(* CODESYS project SLL_Common_exported_from_plc.library
   Title: SLL Common
   CompiledLibraryCompatibilityVersion: CODESYS V3.5 SP16 Patch 5
   DefaultNamespace: SLL_Common
   Version: 0.0.0.1
   Placeholder: SLL_Common
   Company: SLL

Project tree, tasks and I/O mapping:
  libraries: Util, 3.5.19.0 (System); Standard, 3.5.18.0 (System); SysTime, 3.5.17.0 (System); BASIC, 3.3.3.0 (OSCAT)
  Common Control/
    Convert/
    PID/
    Selectors/
    SCALING/
      Stuctures/
      Function Blocks/
      Functions/
  Common Control/
    PID/
      function block Control_PI_Basic [ST]
      data type PID_Settings_Basic
  Convert/
    Functions/
      function TIME_Dword_To_Secs [ST]
      function TIME_Dword_To_Mins [ST]
  SCALING/
    Stuctures/
      data type DUT_SENSOR_SCALE_DWORD_IN_REAL_OUT
      data type DUT_SENSOR_SCALE_REAL_IN_REAL_OUT
      data type DUT_SENSOR_SCALE_WORD_IN_REAL_OUT
      data type DUT_SENSOR_SCALE_DINT_TO_REAL
      data type Union_SensorStatusBits
      data type DUT_SensorStatusBits
    Function Blocks/
      function block Sensor_Scale_Real_To_Real_Struct [FBD]
      function block Sensor_Scale_Dint_To_Real [FBD]
    Functions/
  HMI/
    Functions/
      function HMI_Time_Remain_HHMMSS [ST]
      function HMI_Bool_To_Enable [ST]
      function HMI_Concat_Units [ST]
      function HMI_Sensor_Byte_String [ST]
  SIM/
    function block SIM_Bool [FBD]
    function block SIM_Uint [FBD]
    function block SIM_Byte [FBD]
    function block SIM_Real [FBD]
    function block SIM_Word [FBD]
  STATS/
    function block Cycle_Freq [FBD]
    function block Timestamp_TO [FBD]
    function block Operated_Time_Hours [FBD]
    function block Operated_Time_Min [FBD]
    function block Operated_Time_Sec [FBD]
    function block Cycle_Freq_REAL [FBD]
  SEL/
    function block SEL_Bumpless_Word [FBD]
    function block SEL_Bumpless_Real [FBD]
    function block SEL_Bumpless_Bool [FBD]
    function block SEL_Bumpless_Byte [FBD]
  TIMERS/
    function block DUTY_CYCLE [FBD]
  INPUT/
    function block SWITCH_DEBOUNCE [FBD]
*)

// Common Control/PID/PID_Settings_Basic
TYPE PID_Settings_Basic :
STRUCT
	SUP : REAL;
	OFS : REAL;
	KP : REAL;
	TN : REAL;
	TV : REAL;
	LL : REAL;
	LH : REAL;
	NAME:STRING(20);
END_STRUCT
END_TYPE

// SCALING/Stuctures/DUT_SENSOR_SCALE_DWORD_IN_REAL_OUT
TYPE DUT_SENSOR_SCALE_DWORD_IN_REAL_OUT :
STRUCT
	RAW_UNDER_RANGE:DWORD;	
	RAW_MIN:DWORD;
	RAW_MAX:DWORD;
	RAW_OVER_RANGE:DWORD;
	SCL_MIN:REAL;
	SCL_MAX:REAL;
	BYPASS:BOOL:=0;
	BYPASS_SCL:DWORD:=0;	
END_STRUCT
END_TYPE

// SCALING/Stuctures/DUT_SENSOR_SCALE_REAL_IN_REAL_OUT
TYPE DUT_SENSOR_SCALE_REAL_IN_REAL_OUT :
STRUCT
	RAW_UNDER_RANGE:REAL;	
	RAW_MIN:REAL;
	RAW_MAX:REAL;
	RAW_OVER_RANGE:REAL;
	SCL_MIN:REAL;
	SCL_MAX:REAL;
	BYPASS:BOOL:=0;
	BYPASS_SCL:REAL:=0;		
END_STRUCT
END_TYPE

// SCALING/Stuctures/DUT_SENSOR_SCALE_WORD_IN_REAL_OUT
TYPE DUT_SENSOR_SCALE_WORD_IN_REAL_OUT :
STRUCT
	RAW_UNDER_RANGE:WORD;	
	RAW_MIN:WORD;
	RAW_MAX:WORD;
	RAW_OVER_RANGE:WORD;
	SCL_MIN:REAL;
	SCL_MAX:REAL;
	BYPASS:BOOL:=0;
	BYPASS_SCL:WORD:=0;
	NAME: STRING(20);
	UNITS: STRING(10);
END_STRUCT
END_TYPE

// SCALING/Stuctures/DUT_SENSOR_SCALE_DINT_TO_REAL
TYPE DUT_SENSOR_SCALE_DINT_TO_REAL :
STRUCT
	RAW:DINT;
	RAW_UNDER_RANGE:DINT;	
	RAW_MIN:DINT;
	RAW_MAX:DINT;
	RAW_OVER_RANGE:DINT;
	SCL_MIN:REAL;
	SCL_MAX:REAL;
	BYPASS:BOOL:=0;
	BYPASS_SCL:REAL:=0;
	NAME: STRING(20);
	UNITS: STRING(10);

	SCL:REAL;
	HEALTHY:BOOL;
	UNDER_RANGE:BOOL;
	OVER_RANGE:BOOL;
	STATUS_BYTE:BYTE;	

	RAW_RANGE: REAL;
	SCL_RANGE: REAL;
	RATIO: REAL;	
END_STRUCT
END_TYPE

// SCALING/Stuctures/Union_SensorStatusBits
TYPE Union_SensorStatusBits :
UNION
	bits_:DUT_SensorStatusBits;
	word_:WORD;
	bytes_:ARRAY[0..1] OF BYTE;
END_UNION
END_TYPE

// SCALING/Stuctures/DUT_SensorStatusBits
TYPE DUT_SensorStatusBits :
STRUCT
	HEALTHY:BIT;
	UNDER_RANGE:BIT;
	OVER_RANGE:BIT;
	Spare_B03:BIT;
	Input_Error:BIT;
	ConfigDiagProt_Error:BIT;
	ConfigDiagLevel_Error:BIT;
	Spare_B07:BIT;
	Spare_B08:BIT;
	Spare_B09:BIT;
	Spare_B10:BIT;
	Spare_B11:BIT;
	Spare_B12:BIT;
	Spare_B13:BIT;
	Spare_B14:BIT;
	Spare_B15:BIT;
END_STRUCT
END_TYPE

// Convert/Functions/TIME_Dword_To_Secs
FUNCTION TIME_Dword_To_Secs : TIME
VAR_INPUT
	SECS:DWORD;
END_VAR
VAR
END_VAR

TIME_Dword_To_Secs:=DWORD_TO_TIME(SECS*1000);

END_FUNCTION

// Convert/Functions/TIME_Dword_To_Mins
FUNCTION TIME_Dword_To_Mins : TIME
VAR_INPUT
	MINS:DWORD;
END_VAR
VAR
END_VAR

TIME_Dword_To_Mins:=DWORD_TO_TIME(MINS*60*1000);

END_FUNCTION

// Common Control/PID/Control_PI_Basic
FUNCTION_BLOCK Control_PI_Basic
VAR_INPUT
	ACT : REAL;
	SET : REAL;
	M_I : REAL;
	MAN : BOOL;
	RST : BOOL;
	
	SETTINGS:PID_Settings_Basic;
END_VAR
VAR_OUTPUT
	Y : REAL;
	DIFF : REAL;
	LIM : BOOL;
END_VAR
VAR
	pid : OSCAT_BASIC.FT_PIDWL;
	co : OSCAT_BASIC.CTRL_OUT;
END_VAR

DIFF := OSCAT_BASIC.CTRL_IN(SET, ACT, SETTINGS.SUP);
pid(in := DIFF, kp := SETTINGS.KP, tn := SETTINGS.TN, tv := SETTINGS.TV, lim_l := SETTINGS.LL, lim_h := SETTINGS.LH, rst := RST);
co(ci := pid.Y, OFFSET := SETTINGS.OFS, man_in := M_I, lim_l := SETTINGS.LL, lim_h := SETTINGS.LH, MANUAL := MAN);
Y := co.Y;
LIM := co.LIM;



(* revision history
based on the oscat CTRL_PI with structs to move the settings around more easily
*)

END_FUNCTION_BLOCK

// SEL/SEL_Bumpless_Word
FUNCTION_BLOCK SEL_Bumpless_Word
VAR_INPUT
	G:BOOL;
	AUTO_In0:WORD;
END_VAR
VAR_OUTPUT
	OUT: WORD;
END_VAR
VAR
	G_PREV:BOOL;
END_VAR

VAR_IN_OUT
	MAN_In1: WORD;
END_VAR
VAR // added by the converter: edge detectors and wires of the graphical bodies
    _rt1 : R_TRIG;
END_VAR

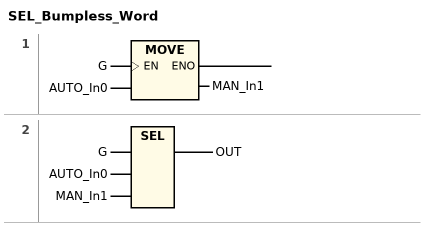
// NETWORK 1
_rt1(CLK := G);
IF _rt1.Q THEN MAN_In1 := AUTO_In0; END_IF

// NETWORK 2
OUT := SEL(G, AUTO_In0, MAN_In1);

END_FUNCTION_BLOCK

// SEL/SEL_Bumpless_Real
FUNCTION_BLOCK SEL_Bumpless_Real
VAR_INPUT
	G:BOOL;
	AUTO_In0:REAL;
END_VAR
VAR_OUTPUT
	OUT: REAL;
END_VAR
VAR
	G_PREV:BOOL;
END_VAR

VAR_IN_OUT
	MAN_In1: REAL;
END_VAR
VAR // added by the converter: edge detectors and wires of the graphical bodies
    _rt1 : R_TRIG;
END_VAR

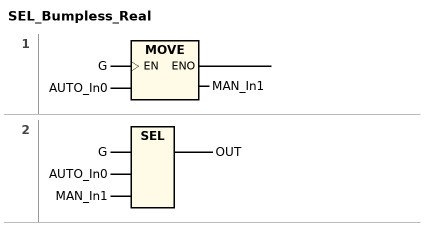
// NETWORK 1
_rt1(CLK := G);
IF _rt1.Q THEN MAN_In1 := AUTO_In0; END_IF

// NETWORK 2
OUT := SEL(G, AUTO_In0, MAN_In1);

END_FUNCTION_BLOCK

// SCALING/Function Blocks/Sensor_Scale_Real_To_Real_Struct
FUNCTION_BLOCK Sensor_Scale_Real_To_Real_Struct
VAR_INPUT
	RAW:REAL;
	SETTINGS:DUT_SENSOR_SCALE_REAL_IN_REAL_OUT;
END_VAR
VAR_OUTPUT
	SCL:REAL;
	HEALTHY:BOOL;
	UNDER_RANGE:BOOL;
	OVER_RANGE:BOOL;	
END_VAR
VAR
	RAW_RANGE: REAL;
	SCL_RANGE: REAL;
	RATIO: REAL;
	PERCENT: REAL;
	PERCENT_INV: REAL;		
END_VAR

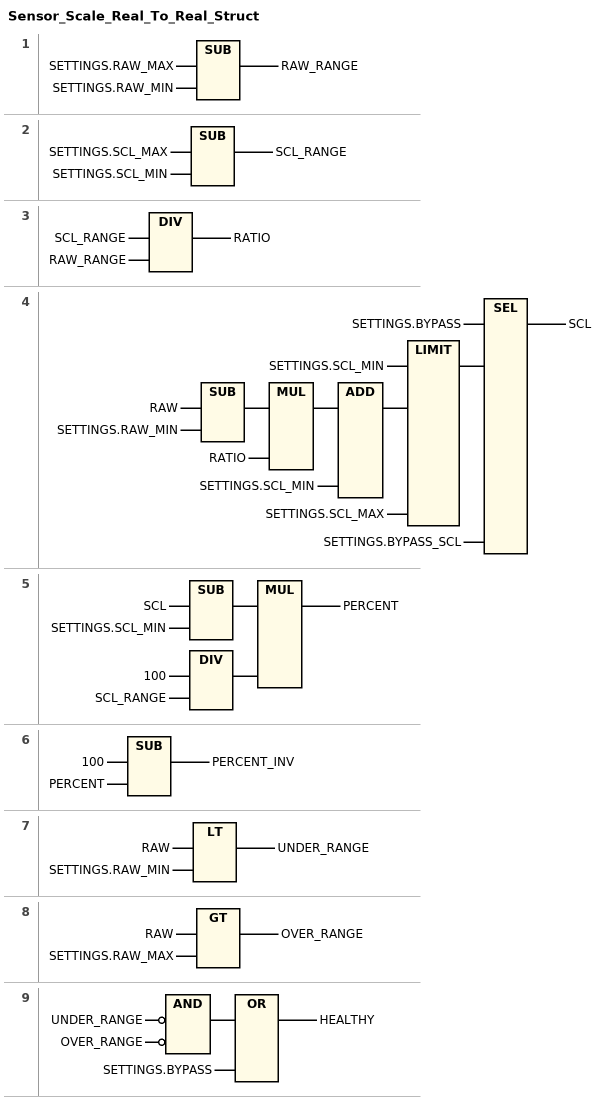
// NETWORK 1
RAW_RANGE := SETTINGS.RAW_MAX - SETTINGS.RAW_MIN;

// NETWORK 2
SCL_RANGE := SETTINGS.SCL_MAX - SETTINGS.SCL_MIN;

// NETWORK 3
RATIO := SCL_RANGE / RAW_RANGE;

// NETWORK 4
SCL := SEL(SETTINGS.BYPASS, LIMIT(SETTINGS.SCL_MIN, (RAW - SETTINGS.RAW_MIN) * RATIO + SETTINGS.SCL_MIN, SETTINGS.SCL_MAX), SETTINGS.BYPASS_SCL);

// NETWORK 5
PERCENT := (SCL - SETTINGS.SCL_MIN) * (100 / SCL_RANGE);

// NETWORK 6
PERCENT_INV := 100 - PERCENT;

// NETWORK 7
UNDER_RANGE := RAW < SETTINGS.RAW_MIN;

// NETWORK 8
OVER_RANGE := RAW > SETTINGS.RAW_MAX;

// NETWORK 9
HEALTHY := NOT UNDER_RANGE AND NOT OVER_RANGE OR SETTINGS.BYPASS;

END_FUNCTION_BLOCK

// SCALING/Function Blocks/Sensor_Scale_Dint_To_Real
FUNCTION_BLOCK Sensor_Scale_Dint_To_Real
VAR_INPUT
	RAW:DINT;
	RAW_UNDER_RANGE:DINT;	
	RAW_MIN:DINT;
	RAW_MAX:DINT;
	RAW_OVER_RANGE:DINT;
	SCL_MIN:REAL;
	SCL_MAX:REAL;
	BYPASS:BOOL:=0;
	BYPASS_SCL:REAL:=0;
	NAME: STRING(30);
	UNITS: STRING(10);
END_VAR
VAR_OUTPUT
	SCL:REAL;
	HEALTHY:BOOL;
	UNDER_RANGE:BOOL;
	OVER_RANGE:BOOL;
	STATUS_BYTE:BYTE;	
END_VAR
VAR
	RAW_RANGE: REAL;
	SCL_RANGE: REAL;
	RATIO: REAL;
	PERCENT: REAL;
	PERCENT_INV: REAL;			
END_VAR

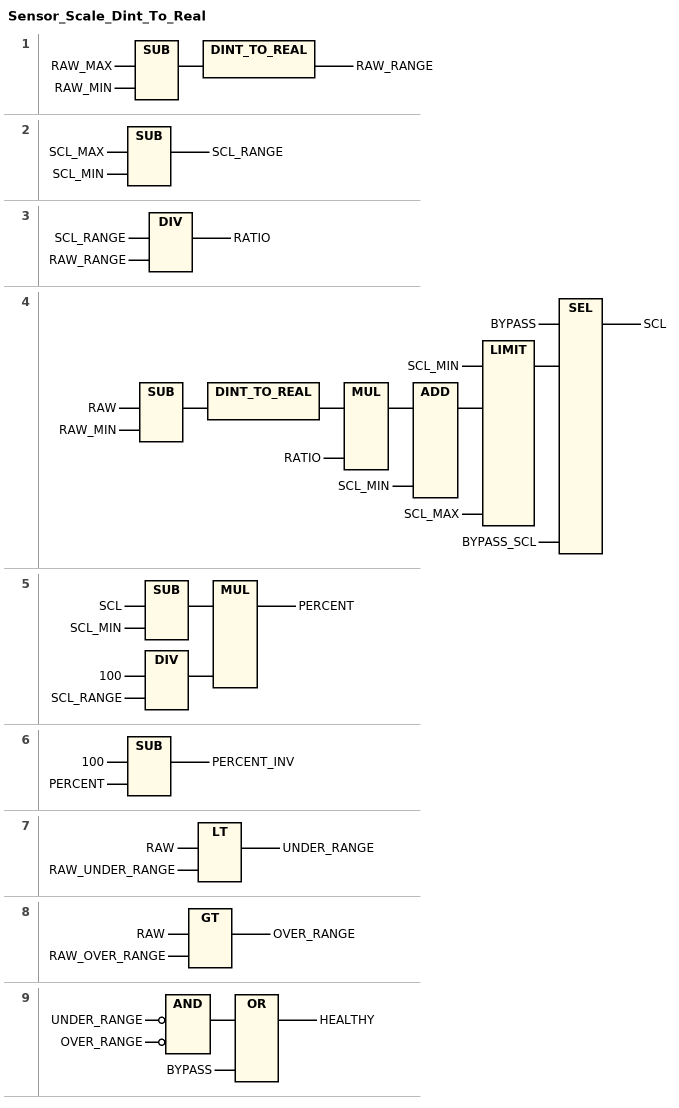
// NETWORK 1
RAW_RANGE := DINT_TO_REAL(RAW_MAX - RAW_MIN);

// NETWORK 2
SCL_RANGE := SCL_MAX - SCL_MIN;

// NETWORK 3
RATIO := SCL_RANGE / RAW_RANGE;

// NETWORK 4
SCL := SEL(BYPASS, LIMIT(SCL_MIN, DINT_TO_REAL(RAW - RAW_MIN) * RATIO + SCL_MIN, SCL_MAX), BYPASS_SCL);

// NETWORK 5
PERCENT := (SCL - SCL_MIN) * (100 / SCL_RANGE);

// NETWORK 6
PERCENT_INV := 100 - PERCENT;

// NETWORK 7
UNDER_RANGE := RAW < RAW_UNDER_RANGE;

// NETWORK 8
OVER_RANGE := RAW > RAW_OVER_RANGE;

// NETWORK 9
HEALTHY := NOT UNDER_RANGE AND NOT OVER_RANGE OR BYPASS;

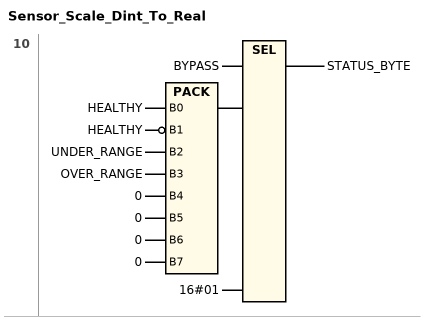
// NETWORK 10
STATUS_BYTE := SEL(BYPASS, PACK(B0 := HEALTHY, B1 := NOT HEALTHY, B2 := UNDER_RANGE, B3 := OVER_RANGE, B4 := 0, B5 := 0, B6 := 0, B7 := 0), 16#01);

END_FUNCTION_BLOCK

// HMI/Functions/HMI_Time_Remain_HHMMSS
FUNCTION HMI_Time_Remain_HHMMSS : STRING
VAR_INPUT
	In:TIME;
END_VAR
VAR
	Total_ms:DWORD;
	TotalSeconds: DWORD;
	Hours: DWORD;
	Mins: DWORD;
	Secs: DWORD;
	
	Temp_STR:STRING;
	TotalMinutes: DWORD;
END_VAR

Total_ms:=TIME_TO_DWORD(In);

// we just want seconds..
TotalSeconds:=Total_ms/1000;
TotalMinutes:=(TotalSeconds MOD (24*60*60))/60;

Hours:=TotalSeconds/(60*60);
Mins:=(TotalSeconds MOD (60*60))/60;
Secs:=TotalSeconds MOD 60;

Temp_STR:= '';

IF Hours > 0 THEN
	Temp_STR:= CONCAT(Temp_STR,DWORD_TO_STRING(Hours));
	Temp_STR:= CONCAT(Temp_STR,'h');
	Temp_STR:= CONCAT(Temp_STR,DWORD_TO_STRING(Mins));
	Temp_STR:= CONCAT(Temp_STR,'m');
	Temp_STR:= CONCAT(Temp_STR,DWORD_TO_STRING(Secs));
	Temp_STR:= CONCAT(Temp_STR,'s');		
ELSIF Mins > 0 THEN
	Temp_STR:= CONCAT(Temp_STR,DWORD_TO_STRING(Mins));
	Temp_STR:= CONCAT(Temp_STR,'m');
	Temp_STR:= CONCAT(Temp_STR,DWORD_TO_STRING(Secs));
	Temp_STR:= CONCAT(Temp_STR,'s');		
ELSIF Secs > 0 THEN
	Temp_STR:= CONCAT(Temp_STR,DWORD_TO_STRING(Secs));
	Temp_STR:= CONCAT(Temp_STR,'s');		
ELSE
	Temp_STR:= CONCAT(Temp_STR,'n/a');	
END_IF;

HMI_Time_Remain_HHMMSS := Temp_STR;

END_FUNCTION

// HMI/Functions/HMI_Bool_To_Enable
FUNCTION HMI_Bool_To_Enable : STRING
VAR_INPUT
	Input:BOOL;
END_VAR
VAR
END_VAR

IF Input THEN
	HMI_Bool_To_Enable:='Enabled';	
ELSE
	HMI_Bool_To_Enable:='Disabled';
END_IF

END_FUNCTION

// HMI/Functions/HMI_Concat_Units
FUNCTION HMI_Concat_Units : STRING
VAR_INPUT
	Input: REAL;
	Units: STRING;	
END_VAR
VAR
	Temp: STRING;
END_VAR

Temp:=REAL_TO_STRING(Input);
Temp:=CONCAT(Temp,' ');
Temp:=CONCAT(Temp,Units);
HMI_Concat_Units:=Temp;

END_FUNCTION

// HMI/Functions/HMI_Sensor_Byte_String
FUNCTION HMI_Sensor_Byte_String : STRING
VAR_INPUT
	Input:BYTE;
END_VAR
VAR
	Temp:STRING;
END_VAR

Temp:='';

IF (Input AND 16#01)<>0 THEN
	Temp:=CONCAT(Temp,'Healthy');
END_IF

IF (Input AND 16#02)<>0 THEN
	Temp:=CONCAT(Temp,'Error');
END_IF

IF (Input AND 16#04)<>0 THEN
	Temp:=CONCAT(Temp,',Under-Range');
END_IF

IF (Input AND 16#08)<>0 THEN
	Temp:=CONCAT(Temp,',Over-Range');
END_IF

HMI_Sensor_Byte_String:=Temp;

END_FUNCTION

// SIM/SIM_Bool
FUNCTION_BLOCK SIM_Bool
VAR_INPUT
	IP_VAL:	 BOOL;
	SIM_ENA: BOOL;
	SIM_VAL: BOOL;
END_VAR
VAR_OUTPUT
	OP_VAL: BOOL;
END_VAR
VAR
END_VAR

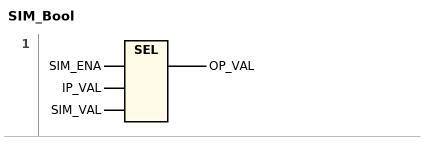
// NETWORK 1
OP_VAL := SEL(SIM_ENA, IP_VAL, SIM_VAL);

END_FUNCTION_BLOCK

// SIM/SIM_Uint
FUNCTION_BLOCK SIM_Uint
VAR_INPUT
	IP_VAL:	 BYTE;
	SIM_ENA: BOOL;
	SIM_VAL: BYTE;
END_VAR
VAR_OUTPUT
	OP_VAL: BYTE;
END_VAR
VAR
END_VAR

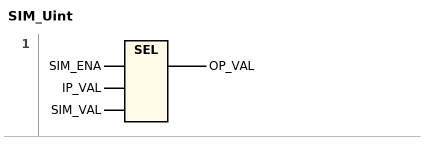
// NETWORK 1
OP_VAL := SEL(SIM_ENA, IP_VAL, SIM_VAL);

END_FUNCTION_BLOCK

// SIM/SIM_Byte
FUNCTION_BLOCK SIM_Byte
VAR_INPUT
	IP_VAL:	 BYTE;
	SIM_ENA: BOOL;
	SIM_VAL: BYTE;
END_VAR
VAR_OUTPUT
	OP_VAL: BYTE;
END_VAR
VAR
END_VAR

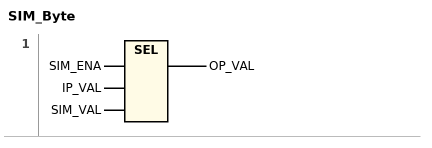
// NETWORK 1
OP_VAL := SEL(SIM_ENA, IP_VAL, SIM_VAL);

END_FUNCTION_BLOCK

// SEL/SEL_Bumpless_Bool
FUNCTION_BLOCK SEL_Bumpless_Bool
VAR_INPUT
	G:BOOL;
	AUTO_In0:BOOL;
END_VAR
VAR_OUTPUT
	OUT: BOOL;
END_VAR
VAR
	G_PREV:BOOL;
END_VAR

VAR_IN_OUT
	MAN_In1: BOOL;
END_VAR
VAR // added by the converter: edge detectors and wires of the graphical bodies
    _rt1 : R_TRIG;
END_VAR

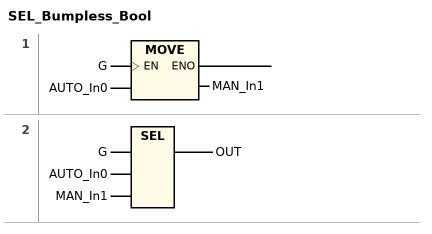
// NETWORK 1
_rt1(CLK := G);
IF _rt1.Q THEN MAN_In1 := AUTO_In0; END_IF

// NETWORK 2
OUT := SEL(G, AUTO_In0, MAN_In1);

END_FUNCTION_BLOCK

// STATS/Cycle_Freq
FUNCTION_BLOCK Cycle_Freq
VAR_INPUT
	READING_INTERVAL_MS:UDINT:=1000;
END_VAR
VAR_OUTPUT
	CYCLES_FREQ:UDINT;
END_VAR
VAR
	CYCLES: UDINT;
	TON_0: TON;
	LAST_READING_MS: UDINT;
END_VAR

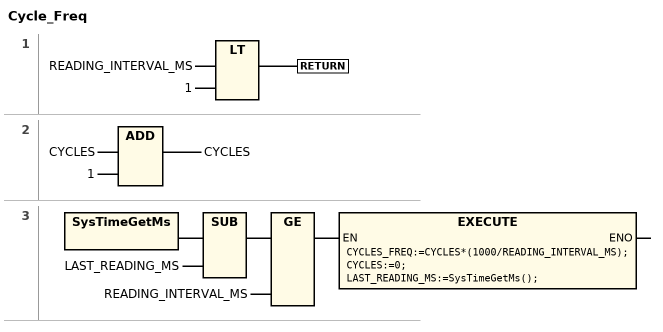
// NETWORK 1
IF READING_INTERVAL_MS < 1 THEN RETURN; END_IF

// NETWORK 2
CYCLES := CYCLES + 1;

// NETWORK 3
IF SysTimeGetMs() - LAST_READING_MS >= READING_INTERVAL_MS THEN
    CYCLES_FREQ:=CYCLES*(1000/READING_INTERVAL_MS);
    CYCLES:=0;
    LAST_READING_MS:=SysTimeGetMs();
END_IF

END_FUNCTION_BLOCK

// STATS/Timestamp_TO
FUNCTION_BLOCK Timestamp_TO
VAR_INPUT
	ENA:BOOL;
	STAMP:BOOL;
	TIMEOUT_MS:UDINT;
	RESET:BOOL;
END_VAR
VAR_OUTPUT
	TIMEOUT:BOOL;
	DIFF:UDINT;
	STAMP_COUNTER:WORD;
	TO_COUNTER:WORD;	
END_VAR
VAR
	TON_0: TON;
	LAST_EVENT_MS: UDINT;
END_VAR
VAR // added by the converter: edge detectors and wires of the graphical bodies
    _rt1 : R_TRIG;
END_VAR

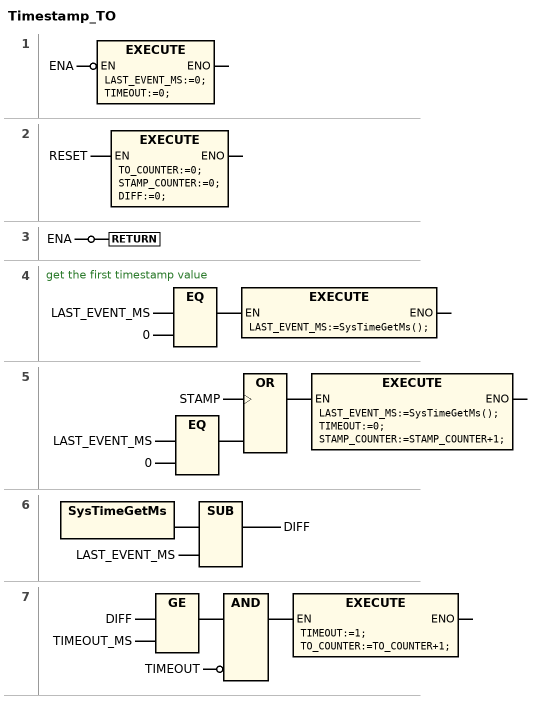
// NETWORK 1
IF NOT ENA THEN
    LAST_EVENT_MS:=0;
    TIMEOUT:=0;
END_IF

// NETWORK 2
IF RESET THEN
    TO_COUNTER:=0;
    STAMP_COUNTER:=0;
    DIFF:=0;
END_IF

// NETWORK 3
IF NOT ENA THEN RETURN; END_IF

// NETWORK 4
// get the first timestamp value
IF LAST_EVENT_MS = 0 THEN LAST_EVENT_MS:=SysTimeGetMs(); END_IF

// NETWORK 5
_rt1(CLK := STAMP);
IF _rt1.Q OR LAST_EVENT_MS = 0 THEN
    LAST_EVENT_MS:=SysTimeGetMs();
    TIMEOUT:=0;
    STAMP_COUNTER:=STAMP_COUNTER+1;
END_IF

// NETWORK 6
DIFF := SysTimeGetMs() - LAST_EVENT_MS;

// NETWORK 7
IF DIFF >= TIMEOUT_MS AND NOT TIMEOUT THEN
    TIMEOUT:=1;
    TO_COUNTER:=TO_COUNTER+1;
END_IF

END_FUNCTION_BLOCK

// STATS/Operated_Time_Hours
FUNCTION_BLOCK Operated_Time_Hours
VAR_INPUT
	Enable: BOOL;
END_VAR
VAR_OUTPUT
	Elapsed_Time: UDINT; // Elapsed time in Hours
END_VAR
VAR
	Stamp: UDINT;
	Current_Time: UDINT;
	Corrected_Time: UDINT;
END_VAR
VAR // added by the converter: edge detectors and wires of the graphical bodies
    _rt1 : R_TRIG;
    _w1 : UDINT;
END_VAR

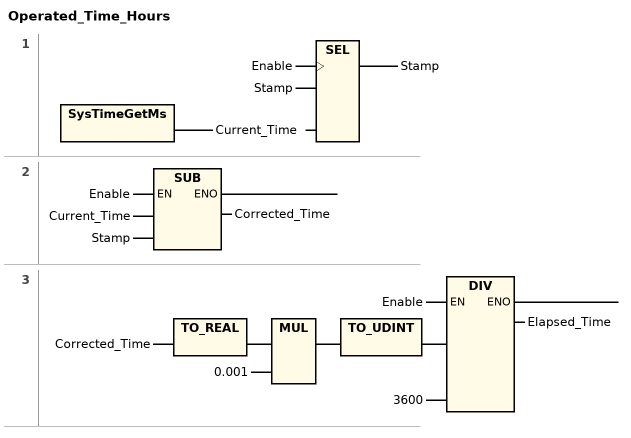
// NETWORK 1
_rt1(CLK := Enable);
_w1 := SysTimeGetMs();
Current_Time := _w1;
Stamp := SEL(_rt1.Q, Stamp, _w1);

// NETWORK 2
IF Enable THEN Corrected_Time := Current_Time - Stamp; END_IF

// NETWORK 3
IF Enable THEN Elapsed_Time := TO_UDINT(TO_REAL(Corrected_Time) * 0.001) / 3600; END_IF

END_FUNCTION_BLOCK

// STATS/Operated_Time_Min
FUNCTION_BLOCK Operated_Time_Min
VAR_INPUT
	Enable: BOOL;
END_VAR
VAR_OUTPUT
	Elapsed_Time: UDINT; // Elapsed time in minutes
END_VAR
VAR
	Stamp: UDINT;
	Current_Time: UDINT;
	Corrected_Time: UDINT;
END_VAR
VAR // added by the converter: edge detectors and wires of the graphical bodies
    _rt1 : R_TRIG;
    _w1 : UDINT;
END_VAR

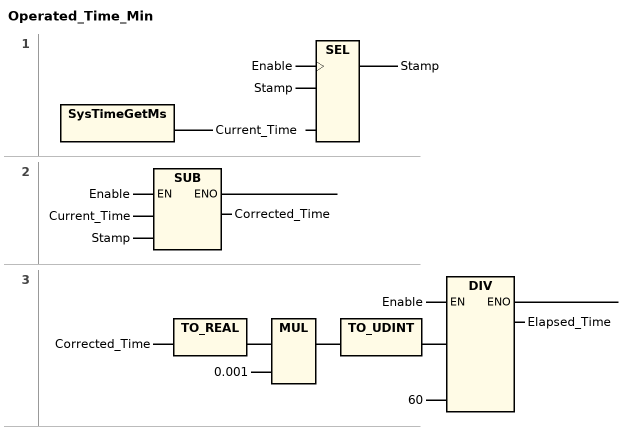
// NETWORK 1
_rt1(CLK := Enable);
_w1 := SysTimeGetMs();
Current_Time := _w1;
Stamp := SEL(_rt1.Q, Stamp, _w1);

// NETWORK 2
IF Enable THEN Corrected_Time := Current_Time - Stamp; END_IF

// NETWORK 3
IF Enable THEN Elapsed_Time := TO_UDINT(TO_REAL(Corrected_Time) * 0.001) / 60; END_IF

END_FUNCTION_BLOCK

// STATS/Operated_Time_Sec
FUNCTION_BLOCK Operated_Time_Sec
VAR_INPUT
	Enable: BOOL;
END_VAR
VAR_OUTPUT
	Elapsed_Time: UDINT; // Elapsed time in seconds
END_VAR
VAR
	Stamp: UDINT;
	Current_Time: UDINT;
	Corrected_Time: UDINT;
END_VAR
VAR // added by the converter: edge detectors and wires of the graphical bodies
    _rt1 : R_TRIG;
    _w1 : UDINT;
END_VAR

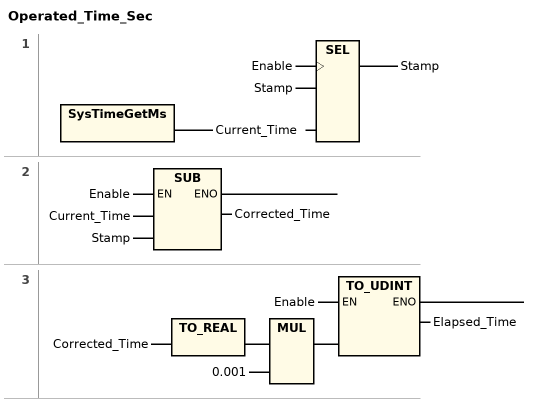
// NETWORK 1
_rt1(CLK := Enable);
_w1 := SysTimeGetMs();
Current_Time := _w1;
Stamp := SEL(_rt1.Q, Stamp, _w1);

// NETWORK 2
IF Enable THEN Corrected_Time := Current_Time - Stamp; END_IF

// NETWORK 3
IF Enable THEN Elapsed_Time := TO_UDINT(TO_REAL(Corrected_Time) * 0.001); END_IF

END_FUNCTION_BLOCK

// SEL/SEL_Bumpless_Byte
FUNCTION_BLOCK SEL_Bumpless_Byte
VAR_INPUT
	G:BOOL;
	AUTO_In0:REAL;
END_VAR
VAR_OUTPUT
	OUT: REAL;
END_VAR
VAR
	G_PREV:BOOL;
END_VAR

VAR_IN_OUT
	MAN_In1: REAL;
END_VAR
VAR // added by the converter: edge detectors and wires of the graphical bodies
    _rt1 : R_TRIG;
END_VAR

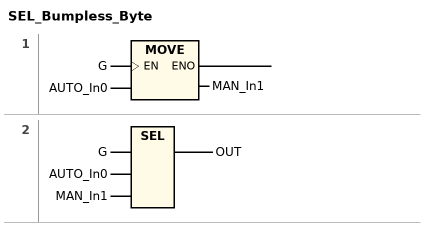
// NETWORK 1
_rt1(CLK := G);
IF _rt1.Q THEN MAN_In1 := AUTO_In0; END_IF

// NETWORK 2
OUT := SEL(G, AUTO_In0, MAN_In1);

END_FUNCTION_BLOCK

// SIM/SIM_Real
FUNCTION_BLOCK SIM_Real
VAR_INPUT
	IP_VAL:	 REAL;
	SIM_ENA: BOOL;
	SIM_VAL: REAL;
END_VAR
VAR_OUTPUT
	OP_VAL: REAL;
END_VAR
VAR
END_VAR

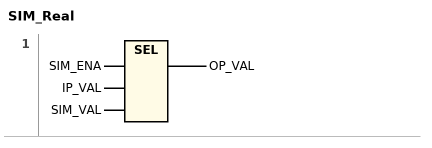
// NETWORK 1
OP_VAL := SEL(SIM_ENA, IP_VAL, SIM_VAL);

END_FUNCTION_BLOCK

// SIM/SIM_Word
FUNCTION_BLOCK SIM_Word
VAR_INPUT
	IP_VAL:	 WORD;
	SIM_ENA: BOOL;
	SIM_VAL: WORD;
END_VAR
VAR_OUTPUT
	OP_VAL: WORD;
END_VAR
VAR
END_VAR

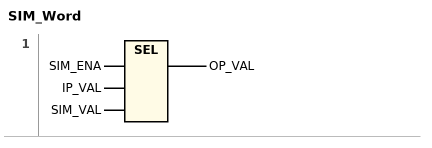
// NETWORK 1
OP_VAL := SEL(SIM_ENA, IP_VAL, SIM_VAL);

END_FUNCTION_BLOCK

// TIMERS/DUTY_CYCLE
FUNCTION_BLOCK DUTY_CYCLE
VAR_INPUT
	IN: BOOL;
	PT_CYCLE: TIME; // Period in TIME
	DUTY: WORD;	// 0-1000 duty (500 = 50%)
END_VAR
VAR_OUTPUT
	Q: BOOL;
END_VAR
VAR
	TON_0: TON;
	PT_ON: TIME;
END_VAR

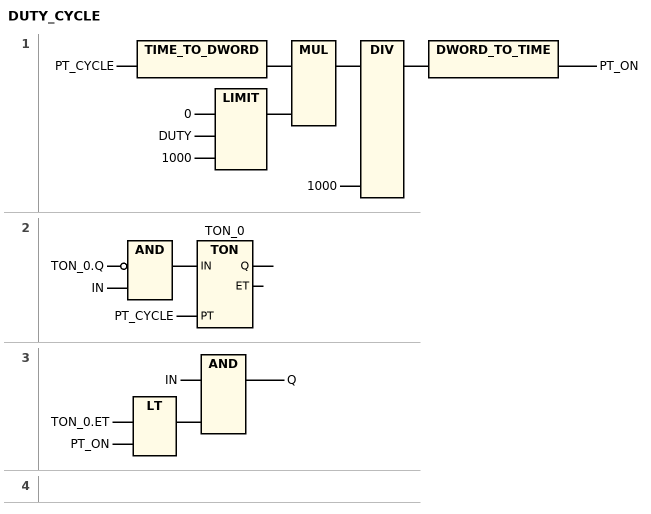
// NETWORK 1
PT_ON := DWORD_TO_TIME((TIME_TO_DWORD(PT_CYCLE) * LIMIT(0, DUTY, 1000)) / 1000);

// NETWORK 2
TON_0(IN := NOT TON_0.Q AND IN, PT := PT_CYCLE); // TON

// NETWORK 3
Q := IN AND TON_0.ET < PT_ON;

// NETWORK 4

END_FUNCTION_BLOCK

// INPUT/SWITCH_DEBOUNCE
FUNCTION_BLOCK SWITCH_DEBOUNCE
VAR_INPUT
	DigIn: BOOL;
	Set_TM: TIME;
	Reset_TM: TIME;	
END_VAR
VAR_OUTPUT
	DigOut: BOOL;
END_VAR
VAR
	Set_TON: TON;
	Reset_TON: TON;
	_SR: SR;
END_VAR

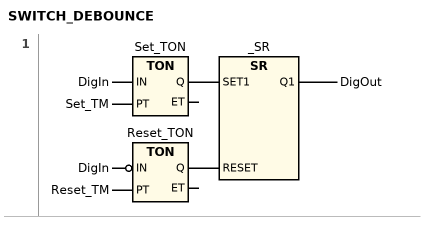
// NETWORK 1
Set_TON(IN := DigIn, PT := Set_TM); // TON
Reset_TON(IN := NOT DigIn, PT := Reset_TM); // TON
_SR(SET1 := Set_TON.Q, RESET := Reset_TON.Q); // SR
DigOut := _SR.Q1;

END_FUNCTION_BLOCK

// STATS/Cycle_Freq_REAL
FUNCTION_BLOCK Cycle_Freq_REAL
VAR_INPUT
	READING_INTERVAL_MS:UDINT:=1000;
END_VAR
VAR_OUTPUT
	CYCLES_FREQ:REAL;
END_VAR
VAR
	CYCLES: REAL;
	TON_0: TON;
	LAST_READING_MS: UDINT;
END_VAR

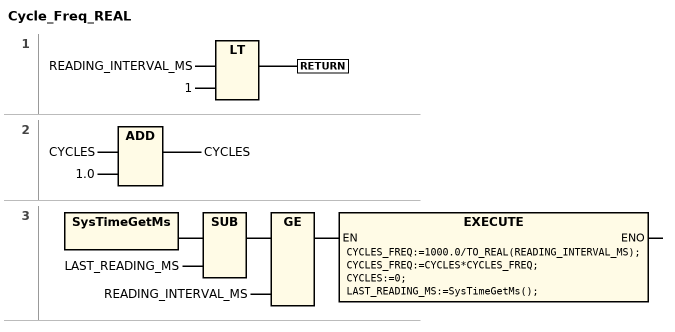
// NETWORK 1
IF READING_INTERVAL_MS < 1 THEN RETURN; END_IF

// NETWORK 2
CYCLES := CYCLES + 1.0;

// NETWORK 3
IF SysTimeGetMs() - LAST_READING_MS >= READING_INTERVAL_MS THEN
    CYCLES_FREQ:=1000.0/TO_REAL(READING_INTERVAL_MS);
    CYCLES_FREQ:=CYCLES*CYCLES_FREQ;
    CYCLES:=0;
    LAST_READING_MS:=SysTimeGetMs();
END_IF

END_FUNCTION_BLOCK
